// TIA Portal V16 export
// export: Created 2024-04-19T14:53:47.1005315Z, ExportSetting WithDefaults, DisplayName Totally Integrated Automation Portal, DisplayVersion V16 Update 6, DisplayName TIA Portal Version Control Interface, DisplayVersion V16 Update 2, DisplayName TIA Portal Openness, DisplayVersion V16 Update 6, DisplayName TIA Portal Test Suite Advanced, DisplayVersion V16, DisplayName SINAMICS Startdrive Advanced, DisplayVersion V16 Update 5, DisplayName SINAMICS Startdrive G130, G150, S120, S150, SINAMICS MV, S210, DisplayVersion V16 Update 5, DisplayName SINAMICS Startdrive G110M, G120, G120C, G120D, G120P, G115D, DisplayVersion V16 Update 5, DisplayName STEP 7 Professional, DisplayVersion V16 Update 6, DisplayName STEP 7 Safety, DisplayVersion V16, DisplayName WinCC Advanced, DisplayVersion V16 Update 6
TYPE "SCA_slatConveyor_IO_Input"
// stored: IsFailsafeCompliant false
   STRUCT
      Safety_switch : Bool;   // Safety switch
      Entry_pec : Bool;   // Entry photocell
      Exit_pec : Bool;   // Exit photocell
      Next_entry_pec : Bool;   // Entry photocell next conveyor
      Prev_exit_pec : Bool;   // Exit photocell previous conveyor
      Man_cnv_fwd : Bool;   // Conveyor manual forward switch
      Man_cnv_rev : Bool;   // Conveyor manual reverse switch
   END_STRUCT;
END_TYPE
